TYPE (* A Template for an Attribute Type *)
  (* Version 0.0, 2023-11-21, 4DIAC-IDE, 4DIAC-Consortium *)
  AttributeDeclaration : STRUCT
    AttributeName : ANY_ELEMENTARY; (* Description *)
  END_STRUCT;
END_TYPE
